# EPICS autosave request: iocBoot/iocrsfsv/auto_settings_rsfsv.req
file "rsfsv_settings.req",                P=$(P),  R=$(R)
